// TIA Portal V19 export
TYPE "Burkett 8691 REV.3"
TITLE = Burkett_Type8691.rev3_Params
// DEVICEID : 2224899    IODD Version 1.3
//  VENDOR : Burkett
// Documentation Version : 1.03
//  DATE: 28.08.2023 
// 
//  Comment : Burkett_Type8691.rev3_Params
   STRUCT
      StandardStructure : Struct
         Header : Struct
            NumberParameter : Int := 24;   // Number of device parameters (Device Identification + Device Parameter)
            AdressParamDownLoad : Int := 20;   // Start adress for ParamDownload signals in this struct
            AdressDeviceIndent : Int := 44;   // Start adress for Device Identification Parameters in this struct (82 Bytes ea)
            AdressApplicSpez : Int := 700;   // Start adress ApplicationSpezificTag (82 Bytes ea) [9]
            AdressDeviceParam : Int := 782;   // Start adress for Device Parameters in this Area (20 Bytes ea) [15]
            AdressKommando : Int := 1082;   // Start adress for Device Commandos
            NumberCommandos : Int := 9;   // Number of Commandos of the device
            Spare01 : Int;   // spare
            Spare02 : Int;   // spare
            Spare03 : Int;   // spare
         END_STRUCT;
         Paramdownload : Struct
            ParamDownLoadStart : Struct   // Parameter Download Start (Only if master and device are V1.1)
               BlockStat : DWord;   // function block status
               IOLStat : DWord;   // IO-Link Status
            END_STRUCT;
            ParamDownLoadEnd : Struct   // Parameter Download End (Only if master and device are V1.1)
               BlockStat : DWord;   // function block status
               IOLStat : DWord;   // IO-Link Status
            END_STRUCT;
            ParamDownLoadStore : Struct   // Parameter Download Store (Only if master and device are V1.1)
               BlockStat : DWord;   // function block status
               IOLStat : DWord;   // IO-Link Status
            END_STRUCT;
         END_STRUCT;
         DeviceIndentification : Struct   // device indentification parameter
            V_VendorName : Struct   // Vendor Name
               Text : String[64];
               Index : Int := 16;   // parameter index
               Subindex : Int;   // parameter subindex
               Length : Int := 64;   // parameter length in BYTE for writing
               BlockStat : DWord;   // function block status
               IOLStat : DWord;   // IO-Link Status
               RelRead : Bool := TRUE;   // reading release
               RelWrite : Bool;   // writing release
            END_STRUCT;
            V_VendorText : Struct   // Vendor Text
               Text : String[64];
               Index : Int := 17;   // parameter index
               Subindex : Int;   // parameter subindex
               Length : Int := 64;   // parameter length in BYTE for writing
               BlockStat : DWord;   // function block status
               IOLStat : DWord;   // IO-Link Status
               RelRead : Bool := TRUE;   // reading release
               RelWrite : Bool;   // writing release
            END_STRUCT;
            V_ProductName : Struct   // Product Name
               Text : String[64];
               Index : Int := 18;   // parameter index
               Subindex : Int;   // parameter subindex
               Length : Int := 64;   // parameter length in BYTE for writing
               BlockStat : DWord;   // function block status
               IOLStat : DWord;   // IO-Link Status
               RelRead : Bool := TRUE;   // reading release
               RelWrite : Bool;   // writing release
            END_STRUCT;
            V_ProductID : Struct   // Product ID
               Text : String[64];
               Index : Int := 19;   // parameter index
               Subindex : Int;   // parameter subindex
               Length : Int := 64;   // parameter length in BYTE for writing
               BlockStat : DWord;   // function block status
               IOLStat : DWord;   // IO-Link Status
               RelRead : Bool := TRUE;   // reading release
               RelWrite : Bool;   // writing release
            END_STRUCT;
            V_ProductText : Struct   // Product Text
               Text : String[64];
               Index : Int := 20;   // parameter index
               Subindex : Int;   // parameter subindex
               Length : Int := 64;   // parameter length in BYTE for writing
               BlockStat : DWord;   // function block status
               IOLStat : DWord;   // IO-Link Status
               RelRead : Bool := TRUE;   // reading release
               RelWrite : Bool;   // writing release
            END_STRUCT;
            V_SerialNumber : Struct   // Serial Number
               Text : String[64];
               Index : Int := 21;   // parameter index
               Subindex : Int;   // parameter subindex
               Length : Int := 16;   // parameter length in BYTE for writing
               BlockStat : DWord;   // function block status
               IOLStat : DWord;   // IO-Link Status
               RelRead : Bool := TRUE;   // reading release
               RelWrite : Bool;   // writing release
            END_STRUCT;
            V_HardwareRevision : Struct   // Hardware Version
               Text : String[64];
               Index : Int := 22;   // parameter index
               Subindex : Int;   // parameter subindex
               Length : Int := 64;   // parameter length in BYTE for writing
               BlockStat : DWord;   // function block status
               IOLStat : DWord;   // IO-Link Status
               RelRead : Bool := TRUE;   // reading release
               RelWrite : Bool;   // writing release
            END_STRUCT;
            V_FirmwareRevision : Struct   // Firmware Version
               Text : String[64];
               Index : Int := 23;   // parameter index
               Subindex : Int;   // parameter subindex
               Length : Int := 64;   // parameter length in BYTE for writing
               BlockStat : DWord;   // function block status
               IOLStat : DWord;   // IO-Link Status
               RelRead : Bool := TRUE;   // reading release
               RelWrite : Bool;   // writing release
            END_STRUCT;
         END_STRUCT;
         ApplicationSpecificTag : Struct   // AppliciationSpecificTag
            V_ApplicationSpecificTa : Struct   // Application Specific Tag
               Text : String[64];
               Index : Int := 24;   // parameter index
               Subindex : Int;   // parameter subindex
               Length : Int := 19;   // parameter length in BYTE for writing
               BlockStat : DWord;   // function block status
               IOLStat : DWord;   // IO-Link Status
               RelRead : Bool := TRUE;   // reading release
               RelWrite : Bool := TRUE;   // writing release
            END_STRUCT;
         END_STRUCT;
         DeviceParameters : Struct   // Device Parameters
            Parameter_01 : Struct   // Switching time monitoring
               Value : Struct   // Opening Time
                  OpeningTime : DInt;   // ms
               END_STRUCT;
               Index : Int := 11278;   // parameter index
               Subindex : Int := 1;   // parameter subindex
               Length : Int := 4;   // parameter length in BYTE for writing
               BlockStat : DWord;   // function block status
               IOLStat : DWord;   // IO-Link Status
               RelRead : Bool := TRUE;   // reading release
               RelWrite : Bool;   // writing release
            END_STRUCT;
            Parameter_02 : Struct   // Switching time monitoring
               Value : Struct   // Closing Time
                  ClosingTime : DInt;   // ms
               END_STRUCT;
               Index : Int := 11278;   // parameter index
               Subindex : Int := 2;   // parameter subindex
               Length : Int := 4;   // parameter length in BYTE for writing
               BlockStat : DWord;   // function block status
               IOLStat : DWord;   // IO-Link Status
               RelRead : Bool := TRUE;   // reading release
               RelWrite : Bool;   // writing release
            END_STRUCT;
            Parameter_03 : Struct   // Totalizer for covered distance
               Value : Struct   // Enable totalizer
                  EnableTotaliser : Byte := BYTE#16#01;   // Disabled = 0. Enabled = 1
                  Byte01 : Byte;
                  Byte02 : Byte;
                  Byte03 : Byte;
               END_STRUCT;
               Index : Int := 11269;   // parameter index
               Subindex : Int := 1;   // parameter subindex
               Length : Int := 1;   // parameter length in BYTE for writing
               BlockStat : DWord;   // function block status
               IOLStat : DWord;   // IO-Link Status
               RelRead : Bool := TRUE;   // reading release
               RelWrite : Bool := TRUE;   // writing release
            END_STRUCT;
            Parameter_04 : Struct   // Totalizer for covered distance
               Value : Struct   // Reset totalizer
                  ResetTotaliser : Byte;   // The reset is triggered by writing 1. The device will reset the value to 0
                  Byte01 : Byte;
                  Byte02 : Byte;
                  Byte03 : Byte;
               END_STRUCT;
               Index : Int := 11269;   // parameter index
               Subindex : Int := 2;   // parameter subindex
               Length : Int := 1;   // parameter length in BYTE for writing
               BlockStat : DWord;   // function block status
               IOLStat : DWord;   // IO-Link Status
               RelRead : Bool := TRUE;   // reading release
               RelWrite : Bool := TRUE;   // writing release
            END_STRUCT;
            Parameter_05 : Struct   // Totalizer for covered distance
               Value : Struct   // Progress Totaliser
                  ProgressTotaliser : Real;   // %
               END_STRUCT;
               Index : Int := 11269;   // parameter index
               Subindex : Int := 3;   // parameter subindex
               Length : Int := 4;   // parameter length in BYTE for writing
               BlockStat : DWord;   // function block status
               IOLStat : DWord;   // IO-Link Status
               RelRead : Bool := TRUE;   // reading release
               RelWrite : Bool;   // writing release
            END_STRUCT;
            Parameter_06 : Struct   // Totalizer for covered distance
               Value : Struct   // Desired interval for maintenance
                  IntervalTotaliser : Real;   // mm
               END_STRUCT;
               Index : Int := 11269;   // parameter index
               Subindex : Int := 4;   // parameter subindex
               Length : Int := 4;   // parameter length in BYTE for writing
               BlockStat : DWord;   // function block status
               IOLStat : DWord;   // IO-Link Status
               RelRead : Bool := TRUE;   // reading release
               RelWrite : Bool := TRUE;   // writing release
            END_STRUCT;
            Parameter_07 : Struct   // Totalizer for covered distance
               Value : Struct   // Totaliser Value to be monitored at time of reset
                  ValueTotaliser : Real;
               END_STRUCT;
               Index : Int := 11269;   // parameter index
               Subindex : Int := 5;   // parameter subindex
               Length : Int := 4;   // parameter length in BYTE for writing
               BlockStat : DWord;   // function block status
               IOLStat : DWord;   // IO-Link Status
               RelRead : Bool := TRUE;   // reading release
               RelWrite : Bool;   // writing release
            END_STRUCT;
            Parameter_08 : Struct   // Totalizer for total valve cycles
               Value : Struct   // Enable totalizer
                  EnableTotaliser : Byte := BYTE#16#01;   // Disabled = 0. Enabled = 1
                  Byte01 : Byte;
                  Byte02 : Byte;
                  Byte03 : Byte;
               END_STRUCT;
               Index : Int := 11270;   // parameter index
               Subindex : Int := 1;   // parameter subindex
               Length : Int := 1;   // parameter length in BYTE for writing
               BlockStat : DWord;   // function block status
               IOLStat : DWord;   // IO-Link Status
               RelRead : Bool := TRUE;   // reading release
               RelWrite : Bool := TRUE;   // writing release
            END_STRUCT;
            Parameter_09 : Struct   // Totalizer for total valve cycles
               Value : Struct   // Reset totalizer
                  ResetTotaliser : Byte;   // The reset is triggered by writing 1. The device will reset the value to 0
                  Byte01 : Byte;
                  Byte02 : Byte;
                  Byte03 : Byte;
               END_STRUCT;
               Index : Int := 11270;   // parameter index
               Subindex : Int := 2;   // parameter subindex
               Length : Int := 1;   // parameter length in BYTE for writing
               BlockStat : DWord;   // function block status
               IOLStat : DWord;   // IO-Link Status
               RelRead : Bool := TRUE;   // reading release
               RelWrite : Bool := TRUE;   // writing release
            END_STRUCT;
            Parameter_10 : Struct   // Totalizer for total valve cycles
               Value : Struct   // Progress Totaliser
                  ProgressTotaliser : Real;   // %
               END_STRUCT;
               Index : Int := 11270;   // parameter index
               Subindex : Int := 3;   // parameter subindex
               Length : Int := 4;   // parameter length in BYTE for writing
               BlockStat : DWord;   // function block status
               IOLStat : DWord;   // IO-Link Status
               RelRead : Bool := TRUE;   // reading release
               RelWrite : Bool;   // writing release
            END_STRUCT;
            Parameter_11 : Struct   // Totalizer for total valve cycles
               Value : Struct   // Desired interval for maintenance
                  IntervalTotaliser : DInt;
               END_STRUCT;
               Index : Int := 11270;   // parameter index
               Subindex : Int := 4;   // parameter subindex
               Length : Int := 4;   // parameter length in BYTE for writing
               BlockStat : DWord;   // function block status
               IOLStat : DWord;   // IO-Link Status
               RelRead : Bool := TRUE;   // reading release
               RelWrite : Bool := TRUE;   // writing release
            END_STRUCT;
            Parameter_12 : Struct   // Totalizer for Totalizer for operating duration
               Value : Struct   // Enable totalizer
                  EnableTotaliser : Byte := BYTE#16#01;   // Disabled = 0. Enabled = 1
                  Byte01 : Byte;
                  Byte02 : Byte;
                  Byte03 : Byte;
               END_STRUCT;
               Index : Int := 11271;   // parameter index
               Subindex : Int := 1;   // parameter subindex
               Length : Int := 1;   // parameter length in BYTE for writing
               BlockStat : DWord;   // function block status
               IOLStat : DWord;   // IO-Link Status
               RelRead : Bool := TRUE;   // reading release
               RelWrite : Bool := TRUE;   // writing release
            END_STRUCT;
            Parameter_13 : Struct   // Totalizer for Totalizer for operating duration
               Value : Struct   // Reset totalizer
                  ResetTotaliser : Byte;   // The reset is triggered by writing 1. The device will reset the value to 0
                  Byte01 : Byte;
                  Byte02 : Byte;
                  Byte03 : Byte;
               END_STRUCT;
               Index : Int := 11271;   // parameter index
               Subindex : Int := 2;   // parameter subindex
               Length : Int := 1;   // parameter length in BYTE for writing
               BlockStat : DWord;   // function block status
               IOLStat : DWord;   // IO-Link Status
               RelRead : Bool := TRUE;   // reading release
               RelWrite : Bool := TRUE;   // writing release
            END_STRUCT;
            Parameter_14 : Struct   // Totalizer for Totalizer for operating duration
               Value : Struct   // Progress Totaliser
                  ProgressTotaliser : Real;   // %
               END_STRUCT;
               Index : Int := 11271;   // parameter index
               Subindex : Int := 3;   // parameter subindex
               Length : Int := 4;   // parameter length in BYTE for writing
               BlockStat : DWord;   // function block status
               IOLStat : DWord;   // IO-Link Status
               RelRead : Bool := TRUE;   // reading release
               RelWrite : Bool;   // writing release
            END_STRUCT;
            Parameter_15 : Struct   // Totalizer for Totalizer for operating duration
               Value : Struct   // Desired interval for maintenance
                  IntervalTotaliser : DInt;   // ms
               END_STRUCT;
               Index : Int := 11271;   // parameter index
               Subindex : Int := 4;   // parameter subindex
               Length : Int := 4;   // parameter length in BYTE for writing
               BlockStat : DWord;   // function block status
               IOLStat : DWord;   // IO-Link Status
               RelRead : Bool := TRUE;   // reading release
               RelWrite : Bool := TRUE;   // writing release
            END_STRUCT;
         END_STRUCT;
         Commando : Struct   // Commandos
            Commando_01 : Struct   // Device Reset
               Value : Byte := BYTE#16#80;   // 128
               Index : Int := 2;   // parameter index
               Subindex : Int;   // parameter subindex
               Length : Int := 1;   // parameter length in BYTE for writing
               BlockStat : DWord;   // function block status
               IOLStat : DWord;   // IO-Link Status
            END_STRUCT;
            Commando_02 : Struct   // Restore factory settings
               Value : Byte := BYTE#16#82;   // 130
               Index : Int := 2;   // parameter index
               Subindex : Int;   // parameter subindex
               Length : Int := 1;   // parameter length in BYTE for writing
               BlockStat : DWord;   // function block status
               IOLStat : DWord;   // IO-Link Status
            END_STRUCT;
            Commando_03 : Struct   // Start automatic Teach-function
               Value : Byte := BYTE#16#A0;   // 160
               Index : Int := 2;   // parameter index
               Subindex : Int;   // parameter subindex
               Length : Int := 1;   // parameter length in BYTE for writing
               BlockStat : DWord;   // function block status
               IOLStat : DWord;   // IO-Link Status
            END_STRUCT;
            Commando_04 : Struct   // Start manual Teach-function
               Value : Byte := BYTE#16#A1;   // 161
               Index : Int := 2;   // parameter index
               Subindex : Int;   // parameter subindex
               Length : Int := 1;   // parameter length in BYTE for writing
               BlockStat : DWord;   // function block status
               IOLStat : DWord;   // IO-Link Status
            END_STRUCT;
            Commando_05 : Struct   // Abort Teach-function
               Value : Byte := BYTE#16#A2;   // 162
               Index : Int := 2;   // parameter index
               Subindex : Int;   // parameter subindex
               Length : Int := 1;   // parameter length in BYTE for writing
               BlockStat : DWord;   // function block status
               IOLStat : DWord;   // IO-Link Status
            END_STRUCT;
            Commando_06 : Struct   // Enable Teach-In-Operation
               Value : Byte := BYTE#16#A3;   // 163
               Index : Int := 2;   // parameter index
               Subindex : Int;   // parameter subindex
               Length : Int := 1;   // parameter length in BYTE for writing
               BlockStat : DWord;   // function block status
               IOLStat : DWord;   // IO-Link Status
            END_STRUCT;
            Commando_07 : Struct   // Disable Teach-In-Operation
               Value : Byte := BYTE#16#A4;   // 164
               Index : Int := 2;   // parameter index
               Subindex : Int;   // parameter subindex
               Length : Int := 1;   // parameter length in BYTE for writing
               BlockStat : DWord;   // function block status
               IOLStat : DWord;   // IO-Link Status
            END_STRUCT;
            Commando_08 : Struct   // Confirm end position 1 (manual teach function)
               Value : Byte := BYTE#16#A5;   // 165
               Index : Int := 2;   // parameter index
               Subindex : Int;   // parameter subindex
               Length : Int := 1;   // parameter length in BYTE for writing
               BlockStat : DWord;   // function block status
               IOLStat : DWord;   // IO-Link Status
            END_STRUCT;
            Commando_09 : Struct   // Confirm end position 2 (manual teach function)
               Value : Byte := BYTE#16#A6;   // 166
               Index : Int := 2;   // parameter index
               Subindex : Int;   // parameter subindex
               Length : Int := 1;   // parameter length in BYTE for writing
               BlockStat : DWord;   // function block status
               IOLStat : DWord;   // IO-Link Status
            END_STRUCT;
         END_STRUCT;
      END_STRUCT;
      spare : Array[1..268] of Byte;
   END_STRUCT;
END_TYPE
